// TIA Portal V17 export
// export: Created 2024-09-02T12:50:18.9599664Z, ExportSetting WithDefaults, DisplayName Totally Integrated Automation Portal, DisplayVersion V17, DisplayName TIA Portal Openness, DisplayVersion V17, DisplayName TIA Portal Version Control Interface, DisplayVersion V17, DisplayName STEP 7 Professional, DisplayVersion V17, DisplayName STEP 7 Safety, DisplayVersion V17, DisplayName WinCC Professional, DisplayVersion V17
FUNCTION "AnwFC_Desoutter_OP70_2" : Void   // FC110, LAD
{ S7_Optimized_Access := 'TRUE' }
VERSION : 0.1
// stored: AutoNumber false, IsIECCheckEnabled false, SetENOAutomatically false, UDAEnableTagReadback false
   VAR_TEMP
      tVKE0 : Bool;
      tVKE1 : Bool;
      tAuto : Bool;
      tHand : Bool;
      Motion_Release : Bool;
      t_dummy : Bool;
      tHmiBld : Bool;
      tHmiEnbl : Bool;
      tProgram_nr : Byte;
      tCnt : Int;
      tBAmode : Int;
      tHmiNr : Int;
      tArray_ID_POP : Array[0..15] of Char;
      Part_ID_Ready : Bool;
      tCnt_char : UInt;
      Position_of_ScrewDriver_Ready : Bool;
      tHmiScreen : Bool;
      tHmiRelease : Bool;
   END_VAR
   VAR_TEMP   // added for the SCL form of the ladder/FBD networks
      _w1 : Bool;
      _w2 : Bool;
   END_VAR
BEGIN

REGION Network 1: ############# Start Up Conditions ###############
END_REGION

REGION Network 2: VKE0/1
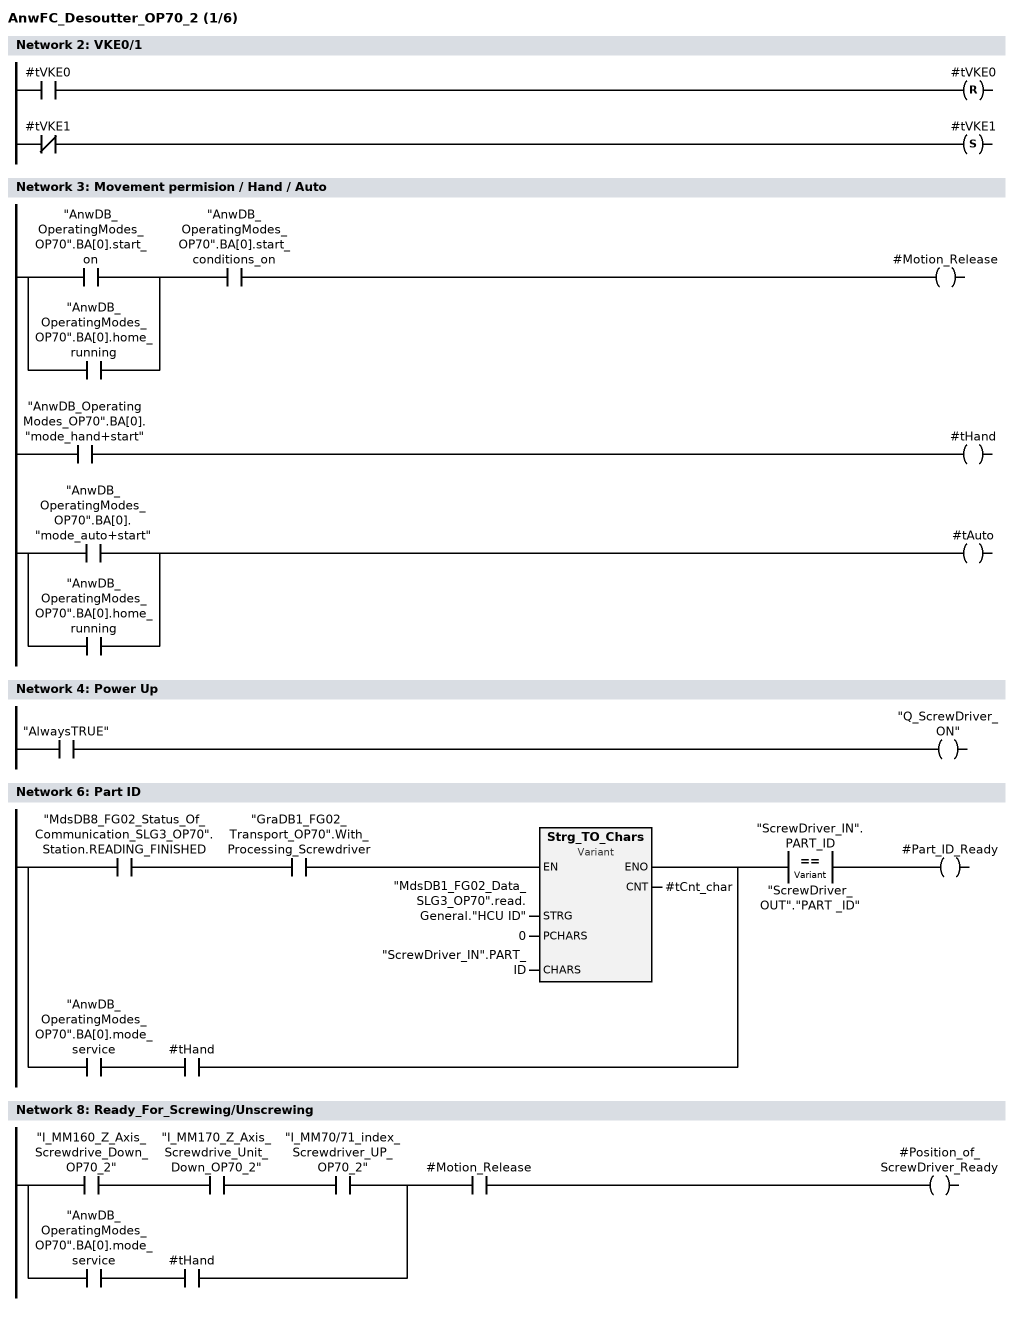
   RUNG wire#powerrail
      Contact( #tVKE0 )
      R_Coil( #tVKE0 )
   END_RUNG
   RUNG wire#powerrail
      I_Contact( #tVKE1 )
      S_Coil( #tVKE1 )
   END_RUNG
   // the same network as SCL:
   IF #tVKE0 THEN #tVKE0 := FALSE; END_IF;
   IF NOT #tVKE1 THEN #tVKE1 := TRUE; END_IF;
END_REGION

REGION Network 3: Movement permision / Hand / Auto
   RUNG wire#powerrail
      Contact( "AnwDB_OperatingModes_OP70".BA[0].start_on )
      wire#w1
      Contact( "AnwDB_OperatingModes_OP70".BA[0].start_conditions_on )
      Coil( #Motion_Release )
   END_RUNG
   RUNG wire#powerrail
      Contact( "AnwDB_OperatingModes_OP70".BA[0].home_running )
   END_RUNG wire#w1
   RUNG wire#powerrail
      Contact( "AnwDB_OperatingModes_OP70".BA[0]."mode_hand+start" )
      Coil( #tHand )
   END_RUNG
   RUNG wire#powerrail
      Contact( "AnwDB_OperatingModes_OP70".BA[0]."mode_auto+start" )
      wire#w2
      Coil( #tAuto )
   END_RUNG
   RUNG wire#powerrail
      Contact( "AnwDB_OperatingModes_OP70".BA[0].home_running )
   END_RUNG wire#w2
   // the same network as SCL:
   #Motion_Release := ("AnwDB_OperatingModes_OP70".BA[0].start_on OR "AnwDB_OperatingModes_OP70".BA[0].home_running) AND "AnwDB_OperatingModes_OP70".BA[0].start_conditions_on;
   #tHand := "AnwDB_OperatingModes_OP70".BA[0]."mode_hand+start";
   #tAuto := "AnwDB_OperatingModes_OP70".BA[0]."mode_auto+start" OR "AnwDB_OperatingModes_OP70".BA[0].home_running;
END_REGION

REGION Network 4: Power Up
   RUNG wire#powerrail
      Contact( "AlwaysTRUE" )
      Coil( "Q_ScrewDriver_ON" )
   END_RUNG
   // the same network as SCL:
   "Q_ScrewDriver_ON" := "AlwaysTRUE";
END_REGION

REGION Network 5: ############# Data Operation ###############
END_REGION

REGION Network 6: Part ID
   RUNG wire#powerrail
      Contact( "MdsDB8_FG02_Status_Of_Communication_SLG3_OP70".Station.READING_FINISHED )
      Contact( "GraDB1_FG02_Transport_OP70".With_Processing_Screwdriver )
      { S7_Templates := "[ptr_type := Variant, strg_type := String]" } Strg_TO_Chars(Strg := "MdsDB1_FG02_Data_SLG3_OP70".read.General."HCU ID", pChars := 0, Chars := "ScrewDriver_IN".PART_ID, Cnt => #tCnt_char)
      wire#w1
      { S7_Templates := "SrcType := Variant" } EQ_Contact(in1 := "ScrewDriver_IN".PART_ID, in2 := "ScrewDriver_OUT"."PART _ID")
      Coil( #Part_ID_Ready )
   END_RUNG
   RUNG wire#powerrail
      Contact( "AnwDB_OperatingModes_OP70".BA[0].mode_service )
      Contact( #tHand )
   END_RUNG wire#w1
   // the same network as SCL:
   #_w1 := "MdsDB8_FG02_Status_Of_Communication_SLG3_OP70".Station.READING_FINISHED AND "GraDB1_FG02_Transport_OP70".With_Processing_Screwdriver;
   Strg_TO_Chars(EN := #_w1,
                 Strg := "MdsDB1_FG02_Data_SLG3_OP70".read.General."HCU ID",
                 pChars := 0,
                 Chars := "ScrewDriver_IN".PART_ID,
                 Cnt => #tCnt_char,
                 ENO => #_w2);
   #Part_ID_Ready := (#_w2 OR ("AnwDB_OperatingModes_OP70".BA[0].mode_service AND #tHand)) AND ("ScrewDriver_IN".PART_ID = "ScrewDriver_OUT"."PART _ID");
END_REGION

REGION Network 7: ############# Program Selection And Start ###############
END_REGION

REGION Network 8: Ready_For_Screwing/Unscrewing
   RUNG wire#powerrail
      Contact( "I_MM160_Z_Axis_Screwdrive_Down_OP70_2" )
      Contact( "I_MM170_Z_Axis_Screwdrive_Unit_Down_OP70_2" )
      Contact( "I_MM70/71_index_Screwdriver_UP_OP70_2" )
      wire#w1
      Contact( #Motion_Release )
      Coil( #Position_of_ScrewDriver_Ready )
   END_RUNG
   RUNG wire#powerrail
      Contact( "AnwDB_OperatingModes_OP70".BA[0].mode_service )
      Contact( #tHand )
   END_RUNG wire#w1
   // the same network as SCL:
   #Position_of_ScrewDriver_Ready := (("I_MM160_Z_Axis_Screwdrive_Down_OP70_2" AND "I_MM170_Z_Axis_Screwdrive_Unit_Down_OP70_2" AND "I_MM70/71_index_Screwdriver_UP_OP70_2") OR ("AnwDB_OperatingModes_OP70".BA[0].mode_service AND #tHand)) AND #Motion_Release;
END_REGION

REGION Network 9: Reset
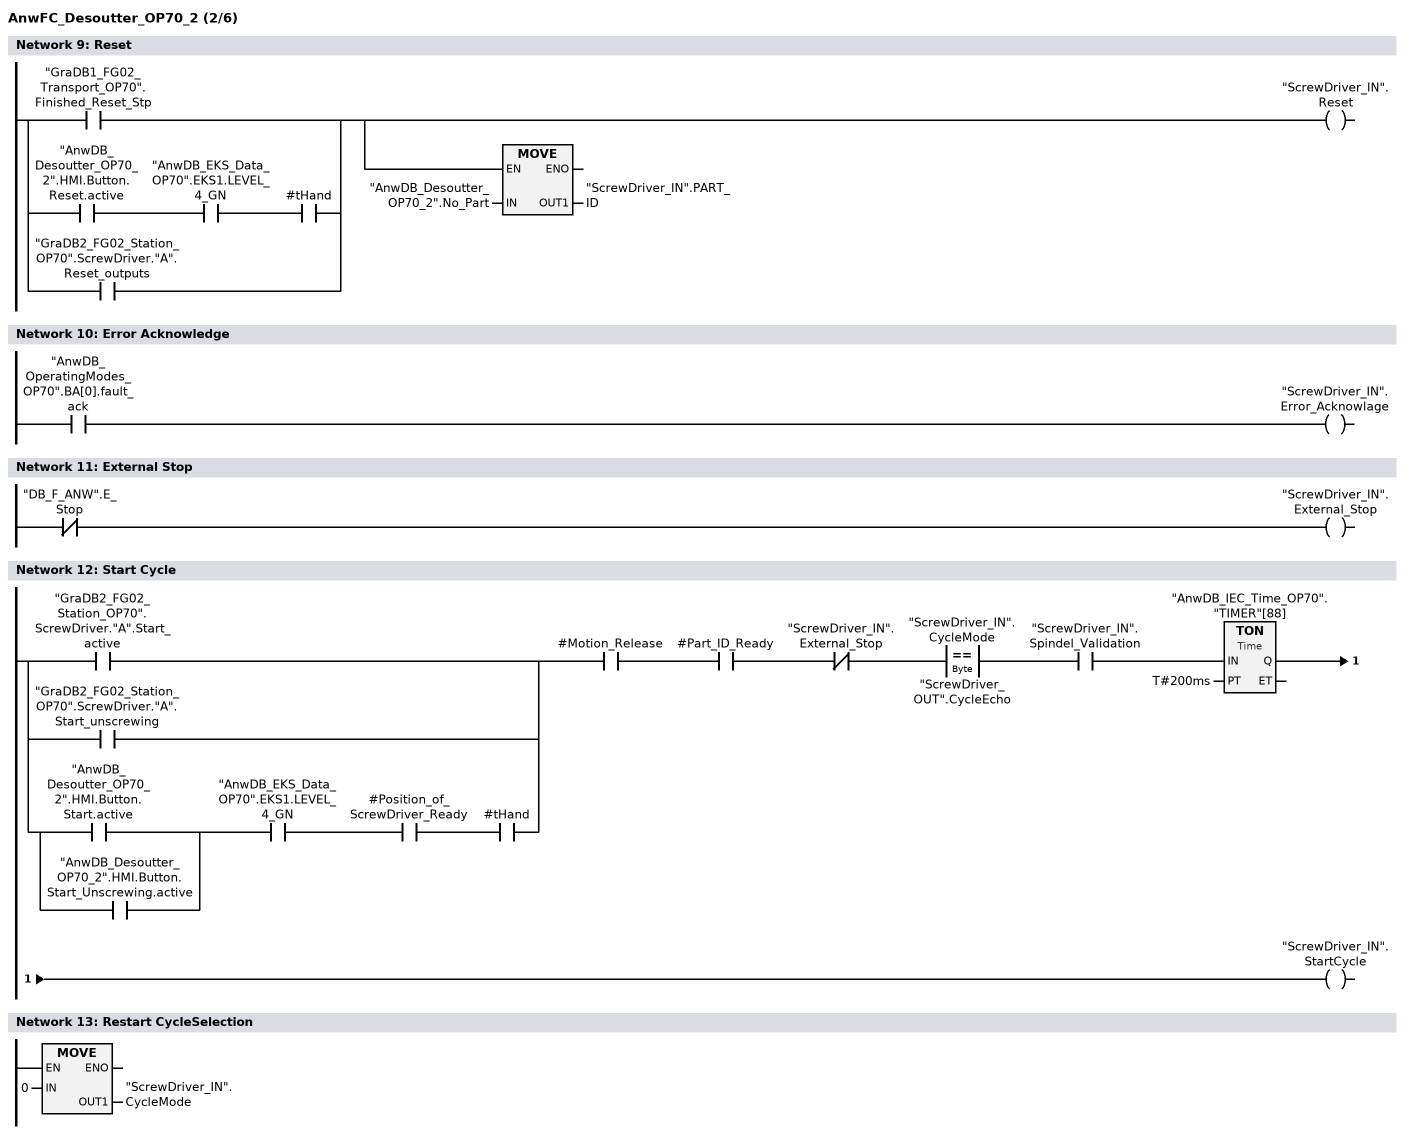
   RUNG wire#powerrail
      Contact( "GraDB1_FG02_Transport_OP70".Finished_Reset_Stp )
      wire#w1
      Coil( "ScrewDriver_IN".Reset )
   END_RUNG
   RUNG wire#powerrail
      Contact( "AnwDB_Desoutter_OP70_2".HMI.Button.Reset.active )
      Contact( "AnwDB_EKS_Data_OP70".EKS1.LEVEL_4_GN )
      Contact( #tHand )
   END_RUNG wire#w1
   RUNG wire#powerrail
      Contact( "GraDB2_FG02_Station_OP70".ScrewDriver."A".Reset_outputs )
   END_RUNG wire#w1
   RUNG wire#w1
      Move(in := "AnwDB_Desoutter_OP70_2".No_Part, out1 => "ScrewDriver_IN".PART_ID)
   END_RUNG
   // the same network as SCL:
   "ScrewDriver_IN".Reset := "GraDB1_FG02_Transport_OP70".Finished_Reset_Stp OR ("AnwDB_Desoutter_OP70_2".HMI.Button.Reset.active AND "AnwDB_EKS_Data_OP70".EKS1.LEVEL_4_GN AND #tHand) OR "GraDB2_FG02_Station_OP70".ScrewDriver."A".Reset_outputs;
   IF "ScrewDriver_IN".Reset THEN "ScrewDriver_IN".PART_ID := "AnwDB_Desoutter_OP70_2".No_Part; END_IF;
END_REGION

REGION Network 10: Error Acknowledge
   RUNG wire#powerrail
      Contact( "AnwDB_OperatingModes_OP70".BA[0].fault_ack )
      Coil( "ScrewDriver_IN".Error_Acknowlage )
   END_RUNG
   // the same network as SCL:
   "ScrewDriver_IN".Error_Acknowlage := "AnwDB_OperatingModes_OP70".BA[0].fault_ack;
END_REGION

REGION Network 11: External Stop
   RUNG wire#powerrail
      I_Contact( "DB_F_ANW".E_Stop )
      Coil( "ScrewDriver_IN".External_Stop )
   END_RUNG
   // the same network as SCL:
   "ScrewDriver_IN".External_Stop := NOT "DB_F_ANW".E_Stop;
END_REGION

REGION Network 12: Start Cycle
   RUNG wire#powerrail
      Contact( "GraDB2_FG02_Station_OP70".ScrewDriver."A".Start_active )
      wire#w1
      Contact( #Motion_Release )
      Contact( #Part_ID_Ready )
      I_Contact( "ScrewDriver_IN".External_Stop )
      { S7_Templates := "SrcType := Byte" } EQ_Contact(in1 := "ScrewDriver_IN".CycleMode, in2 := "ScrewDriver_OUT".CycleEcho)
      Contact( "ScrewDriver_IN".Spindel_Validation )
      { S7_Templates := "time_type := Time" } "AnwDB_IEC_Time_OP70"."TIMER"[88].TON(pt := T#200ms, et =>)
      Coil( "ScrewDriver_IN".StartCycle )
   END_RUNG
   RUNG wire#powerrail
      Contact( "GraDB2_FG02_Station_OP70".ScrewDriver."A".Start_unscrewing )
   END_RUNG wire#w1
   RUNG wire#powerrail
      Contact( "AnwDB_Desoutter_OP70_2".HMI.Button.Start.active )
      wire#w2
      Contact( "AnwDB_EKS_Data_OP70".EKS1.LEVEL_4_GN )
      Contact( #Position_of_ScrewDriver_Ready )
      Contact( #tHand )
   END_RUNG wire#w1
   RUNG wire#powerrail
      Contact( "AnwDB_Desoutter_OP70_2".HMI.Button.Start_Unscrewing.active )
   END_RUNG wire#w2
   // the same network as SCL:
   "AnwDB_IEC_Time_OP70"."TIMER"[88].TON(IN := ("GraDB2_FG02_Station_OP70".ScrewDriver."A".Start_active OR "GraDB2_FG02_Station_OP70".ScrewDriver."A".Start_unscrewing OR (("AnwDB_Desoutter_OP70_2".HMI.Button.Start.active OR "AnwDB_Desoutter_OP70_2".HMI.Button.Start_Unscrewing.active) AND "AnwDB_EKS_Data_OP70".EKS1.LEVEL_4_GN AND #Position_of_ScrewDriver_Ready AND #tHand)) AND #Motion_Release AND #Part_ID_Ready AND NOT "ScrewDriver_IN".External_Stop AND ("ScrewDriver_IN".CycleMode = "ScrewDriver_OUT".CycleEcho) AND "ScrewDriver_IN".Spindel_Validation,
                           PT := T#200ms);
   "ScrewDriver_IN".StartCycle := "AnwDB_IEC_Time_OP70"."TIMER"[88].Q;
END_REGION

REGION Network 13: Restart CycleSelection
   RUNG wire#powerrail
      Move(in := 0, out1 => "ScrewDriver_IN".CycleMode)
   END_RUNG
   // the same network as SCL:
   "ScrewDriver_IN".CycleMode := 0;
END_REGION

REGION Network 14: Cycle Selection - Hand
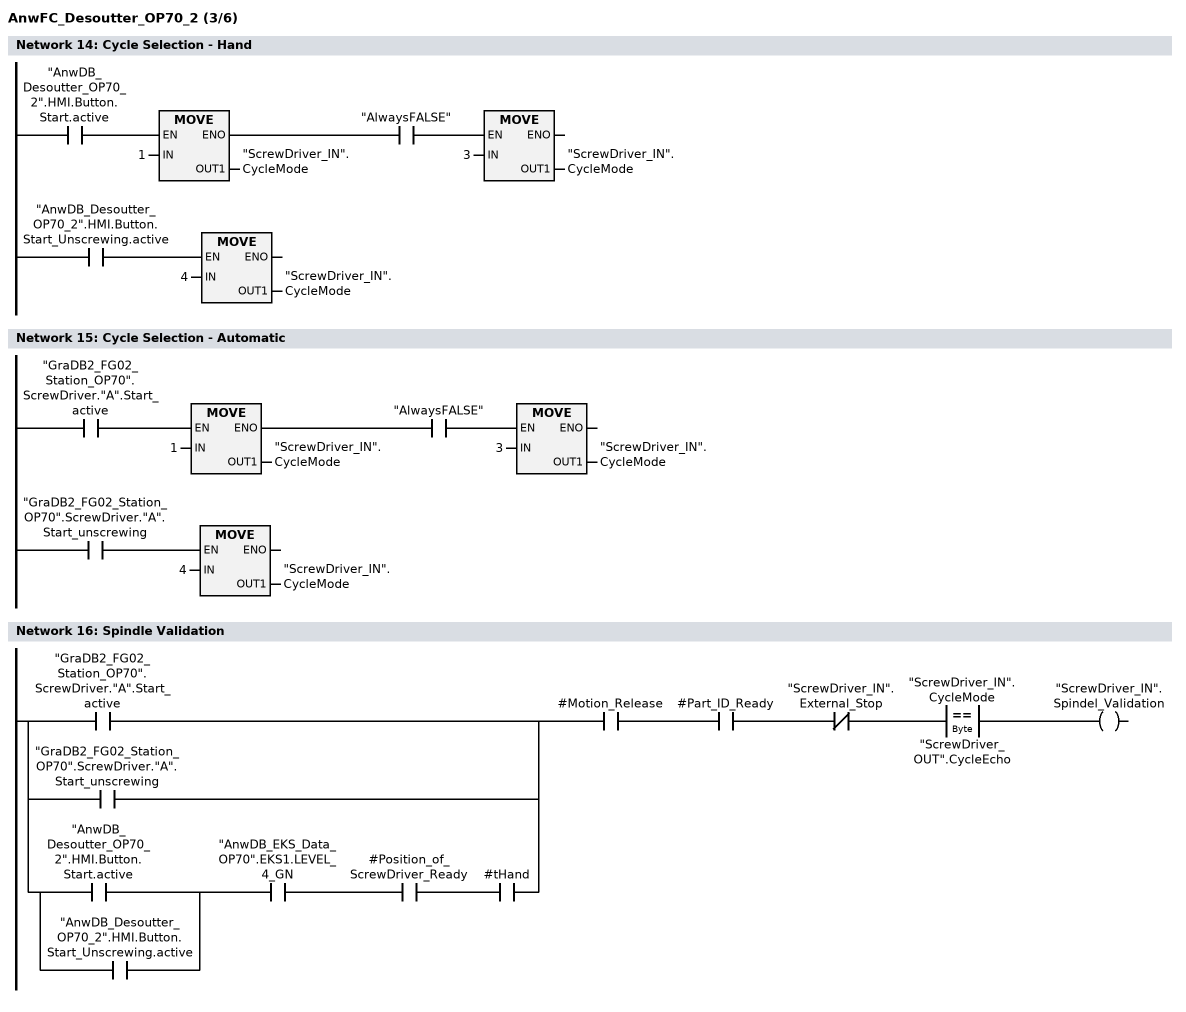
   RUNG wire#powerrail
      Contact( "AnwDB_Desoutter_OP70_2".HMI.Button.Start.active )
      Move(in := 1, out1 => "ScrewDriver_IN".CycleMode)
      Contact( "AlwaysFALSE" )
      Move(in := 3, out1 => "ScrewDriver_IN".CycleMode)
   END_RUNG
   RUNG wire#powerrail
      Contact( "AnwDB_Desoutter_OP70_2".HMI.Button.Start_Unscrewing.active )
      Move(in := 4, out1 => "ScrewDriver_IN".CycleMode)
   END_RUNG
   // the same network as SCL:
   IF "AnwDB_Desoutter_OP70_2".HMI.Button.Start.active THEN "ScrewDriver_IN".CycleMode := 1; END_IF;
   IF "AnwDB_Desoutter_OP70_2".HMI.Button.Start.active AND "AlwaysFALSE" THEN
       "ScrewDriver_IN".CycleMode := 3;
   END_IF;
   IF "AnwDB_Desoutter_OP70_2".HMI.Button.Start_Unscrewing.active THEN
       "ScrewDriver_IN".CycleMode := 4;
   END_IF;
END_REGION

REGION Network 15: Cycle Selection - Automatic
   RUNG wire#powerrail
      Contact( "GraDB2_FG02_Station_OP70".ScrewDriver."A".Start_active )
      Move(in := 1, out1 => "ScrewDriver_IN".CycleMode)
      Contact( "AlwaysFALSE" )
      Move(in := 3, out1 => "ScrewDriver_IN".CycleMode)
   END_RUNG
   RUNG wire#powerrail
      Contact( "GraDB2_FG02_Station_OP70".ScrewDriver."A".Start_unscrewing )
      Move(in := 4, out1 => "ScrewDriver_IN".CycleMode)
   END_RUNG
   // the same network as SCL:
   IF "GraDB2_FG02_Station_OP70".ScrewDriver."A".Start_active THEN "ScrewDriver_IN".CycleMode := 1; END_IF;
   IF "GraDB2_FG02_Station_OP70".ScrewDriver."A".Start_active AND "AlwaysFALSE" THEN
       "ScrewDriver_IN".CycleMode := 3;
   END_IF;
   IF "GraDB2_FG02_Station_OP70".ScrewDriver."A".Start_unscrewing THEN
       "ScrewDriver_IN".CycleMode := 4;
   END_IF;
END_REGION

REGION Network 16: Spindle Validation
   RUNG wire#powerrail
      Contact( "GraDB2_FG02_Station_OP70".ScrewDriver."A".Start_active )
      wire#w1
      Contact( #Motion_Release )
      Contact( #Part_ID_Ready )
      I_Contact( "ScrewDriver_IN".External_Stop )
      { S7_Templates := "SrcType := Byte" } EQ_Contact(in1 := "ScrewDriver_IN".CycleMode, in2 := "ScrewDriver_OUT".CycleEcho)
      Coil( "ScrewDriver_IN".Spindel_Validation )
   END_RUNG
   RUNG wire#powerrail
      Contact( "GraDB2_FG02_Station_OP70".ScrewDriver."A".Start_unscrewing )
   END_RUNG wire#w1
   RUNG wire#powerrail
      Contact( "AnwDB_Desoutter_OP70_2".HMI.Button.Start.active )
      wire#w2
      Contact( "AnwDB_EKS_Data_OP70".EKS1.LEVEL_4_GN )
      Contact( #Position_of_ScrewDriver_Ready )
      Contact( #tHand )
   END_RUNG wire#w1
   RUNG wire#powerrail
      Contact( "AnwDB_Desoutter_OP70_2".HMI.Button.Start_Unscrewing.active )
   END_RUNG wire#w2
   // the same network as SCL:
   "ScrewDriver_IN".Spindel_Validation := ("GraDB2_FG02_Station_OP70".ScrewDriver."A".Start_active OR "GraDB2_FG02_Station_OP70".ScrewDriver."A".Start_unscrewing OR (("AnwDB_Desoutter_OP70_2".HMI.Button.Start.active OR "AnwDB_Desoutter_OP70_2".HMI.Button.Start_Unscrewing.active) AND "AnwDB_EKS_Data_OP70".EKS1.LEVEL_4_GN AND #Position_of_ScrewDriver_Ready AND #tHand)) AND #Motion_Release AND #Part_ID_Ready AND NOT "ScrewDriver_IN".External_Stop AND ("ScrewDriver_IN".CycleMode = "ScrewDriver_OUT".CycleEcho);
END_REGION

REGION Network 17: ############# Program Status ###############
END_REGION

REGION Network 18: BEA[3].Ebit[1] - / BEA[3].Ebit[1] - Searching Program
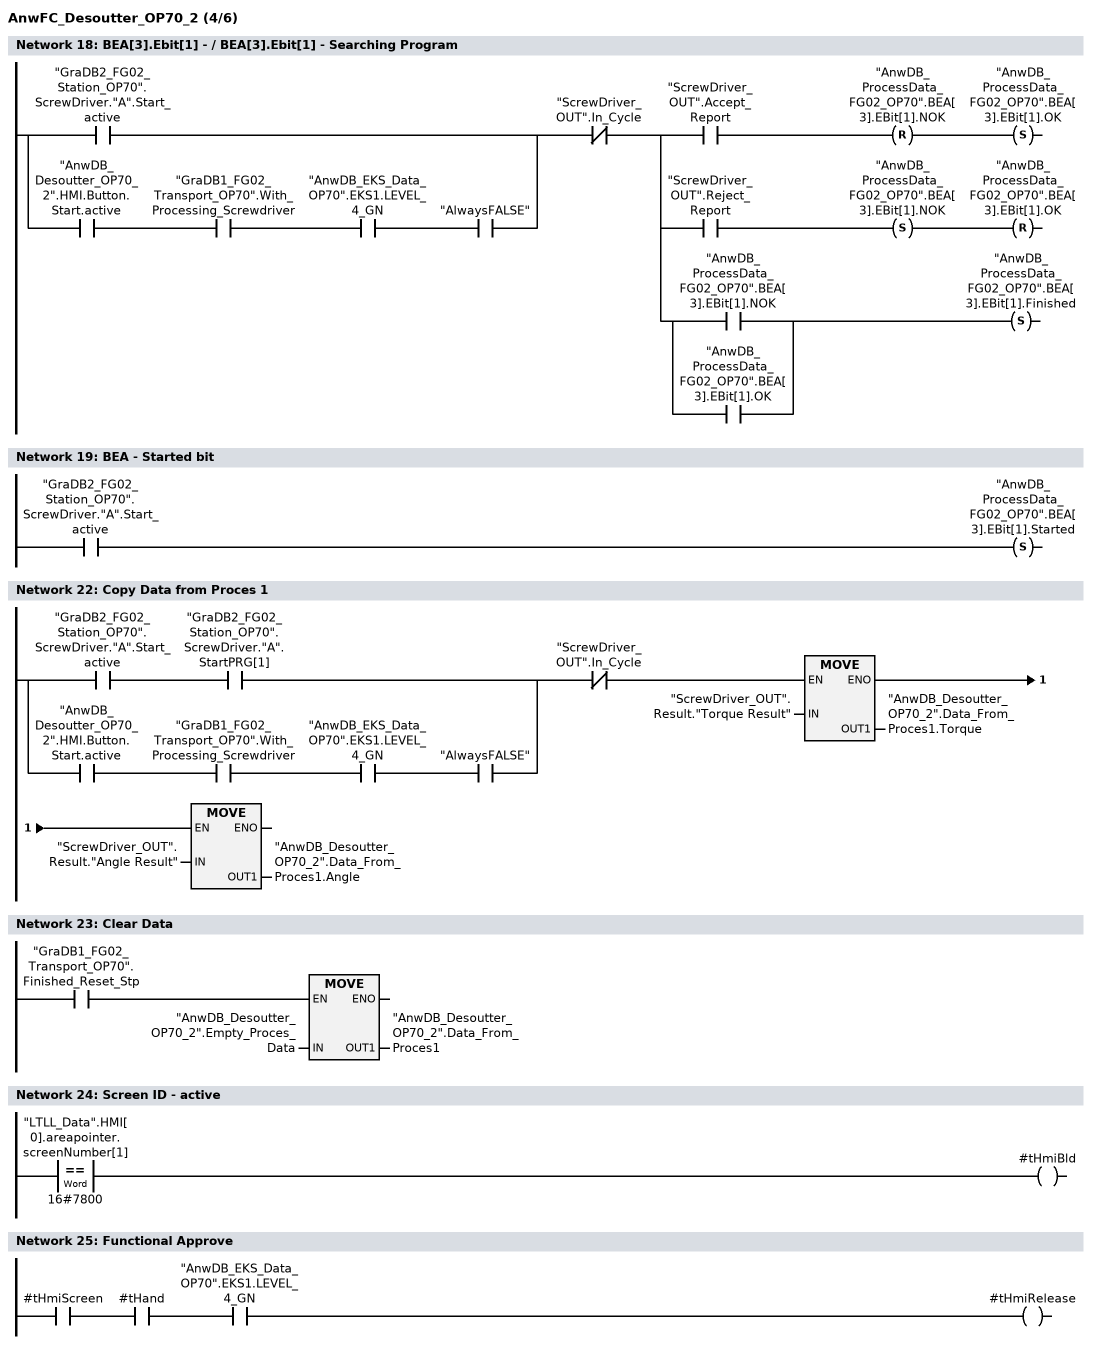
   RUNG wire#powerrail
      Contact( "GraDB2_FG02_Station_OP70".ScrewDriver."A".Start_active )
      wire#w1
      I_Contact( "ScrewDriver_OUT".In_Cycle )
      wire#w2
      Contact( "ScrewDriver_OUT".Accept_Report )
      R_Coil( "AnwDB_ProcessData_FG02_OP70".BEA[3].EBit[1].NOK )
      S_Coil( "AnwDB_ProcessData_FG02_OP70".BEA[3].EBit[1].OK )
   END_RUNG
   RUNG wire#powerrail
      Contact( "AnwDB_Desoutter_OP70_2".HMI.Button.Start.active )
      Contact( "GraDB1_FG02_Transport_OP70".With_Processing_Screwdriver )
      Contact( "AnwDB_EKS_Data_OP70".EKS1.LEVEL_4_GN )
      Contact( "AlwaysFALSE" )
   END_RUNG wire#w1
   RUNG wire#w2
      Contact( "ScrewDriver_OUT".Reject_Report )
      S_Coil( "AnwDB_ProcessData_FG02_OP70".BEA[3].EBit[1].NOK )
      R_Coil( "AnwDB_ProcessData_FG02_OP70".BEA[3].EBit[1].OK )
   END_RUNG
   RUNG wire#w2
      Contact( "AnwDB_ProcessData_FG02_OP70".BEA[3].EBit[1].NOK )
      wire#w3
      S_Coil( "AnwDB_ProcessData_FG02_OP70".BEA[3].EBit[1].Finished )
   END_RUNG
   RUNG wire#w2
      Contact( "AnwDB_ProcessData_FG02_OP70".BEA[3].EBit[1].OK )
   END_RUNG wire#w3
   // the same network as SCL:
   #_w1 := ("GraDB2_FG02_Station_OP70".ScrewDriver."A".Start_active OR ("AnwDB_Desoutter_OP70_2".HMI.Button.Start.active AND "GraDB1_FG02_Transport_OP70".With_Processing_Screwdriver AND "AnwDB_EKS_Data_OP70".EKS1.LEVEL_4_GN AND "AlwaysFALSE")) AND NOT "ScrewDriver_OUT".In_Cycle;
   IF #_w1 AND "ScrewDriver_OUT".Accept_Report THEN
       "AnwDB_ProcessData_FG02_OP70".BEA[3].EBit[1].NOK := FALSE;
       "AnwDB_ProcessData_FG02_OP70".BEA[3].EBit[1].OK := TRUE;
   END_IF;
   IF #_w1 AND "ScrewDriver_OUT".Reject_Report THEN
       "AnwDB_ProcessData_FG02_OP70".BEA[3].EBit[1].NOK := TRUE;
       "AnwDB_ProcessData_FG02_OP70".BEA[3].EBit[1].OK := FALSE;
   END_IF;
   IF #_w1 AND ("AnwDB_ProcessData_FG02_OP70".BEA[3].EBit[1].NOK OR "AnwDB_ProcessData_FG02_OP70".BEA[3].EBit[1].OK) THEN
       "AnwDB_ProcessData_FG02_OP70".BEA[3].EBit[1].Finished := TRUE;
   END_IF;
END_REGION

REGION Network 19: BEA - Started bit
   RUNG wire#powerrail
      Contact( "GraDB2_FG02_Station_OP70".ScrewDriver."A".Start_active )
      S_Coil( "AnwDB_ProcessData_FG02_OP70".BEA[3].EBit[1].Started )
   END_RUNG
   // the same network as SCL:
   IF "GraDB2_FG02_Station_OP70".ScrewDriver."A".Start_active THEN
       "AnwDB_ProcessData_FG02_OP70".BEA[3].EBit[1].Started := TRUE;
   END_IF;
END_REGION

REGION Network 20: ############# HMI ###############
END_REGION

REGION Network 21: ############# Data Copy ###############
END_REGION

REGION Network 22: Copy Data from Proces 1
   RUNG wire#powerrail
      Contact( "GraDB2_FG02_Station_OP70".ScrewDriver."A".Start_active )
      Contact( "GraDB2_FG02_Station_OP70".ScrewDriver."A".StartPRG[1] )
      wire#w1
      I_Contact( "ScrewDriver_OUT".In_Cycle )
      Move(in := "ScrewDriver_OUT".Result."Torque Result", out1 => "AnwDB_Desoutter_OP70_2".Data_From_Proces1.Torque)
      Move(in := "ScrewDriver_OUT".Result."Angle Result", out1 => "AnwDB_Desoutter_OP70_2".Data_From_Proces1.Angle)
   END_RUNG
   RUNG wire#powerrail
      Contact( "AnwDB_Desoutter_OP70_2".HMI.Button.Start.active )
      Contact( "GraDB1_FG02_Transport_OP70".With_Processing_Screwdriver )
      Contact( "AnwDB_EKS_Data_OP70".EKS1.LEVEL_4_GN )
      Contact( "AlwaysFALSE" )
   END_RUNG wire#w1
   // the same network as SCL:
   IF (("GraDB2_FG02_Station_OP70".ScrewDriver."A".Start_active AND "GraDB2_FG02_Station_OP70".ScrewDriver."A".StartPRG[1]) OR ("AnwDB_Desoutter_OP70_2".HMI.Button.Start.active AND "GraDB1_FG02_Transport_OP70".With_Processing_Screwdriver AND "AnwDB_EKS_Data_OP70".EKS1.LEVEL_4_GN AND "AlwaysFALSE")) AND NOT "ScrewDriver_OUT".In_Cycle THEN
       "AnwDB_Desoutter_OP70_2".Data_From_Proces1.Torque := "ScrewDriver_OUT".Result."Torque Result";
       "AnwDB_Desoutter_OP70_2".Data_From_Proces1.Angle := "ScrewDriver_OUT".Result."Angle Result";
   END_IF;
END_REGION

REGION Network 23: Clear Data
   RUNG wire#powerrail
      Contact( "GraDB1_FG02_Transport_OP70".Finished_Reset_Stp )
      Move(in := "AnwDB_Desoutter_OP70_2".Empty_Proces_Data, out1 => "AnwDB_Desoutter_OP70_2".Data_From_Proces1)
   END_RUNG
   // the same network as SCL:
   IF "GraDB1_FG02_Transport_OP70".Finished_Reset_Stp THEN
       "AnwDB_Desoutter_OP70_2".Data_From_Proces1 := "AnwDB_Desoutter_OP70_2".Empty_Proces_Data;
   END_IF;
END_REGION

REGION Network 24: Screen ID - active
   RUNG wire#powerrail
      { S7_Templates := "SrcType := Word" } EQ_Contact(in1 := "LTLL_Data".HMI[0].areapointer.screenNumber[1], in2 := 16#7800)
      Coil( #tHmiBld )
   END_RUNG
   // the same network as SCL:
   #tHmiBld := "LTLL_Data".HMI[0].areapointer.screenNumber[1] = 16#7800;
END_REGION

REGION Network 25: Functional Approve
   RUNG wire#powerrail
      Contact( #tHmiScreen )
      Contact( #tHand )
      Contact( "AnwDB_EKS_Data_OP70".EKS1.LEVEL_4_GN )
      Coil( #tHmiRelease )
   END_RUNG
   // the same network as SCL:
   #tHmiRelease := #tHmiScreen AND #tHand AND "AnwDB_EKS_Data_OP70".EKS1.LEVEL_4_GN;
END_REGION

REGION Network 26: Available of Button
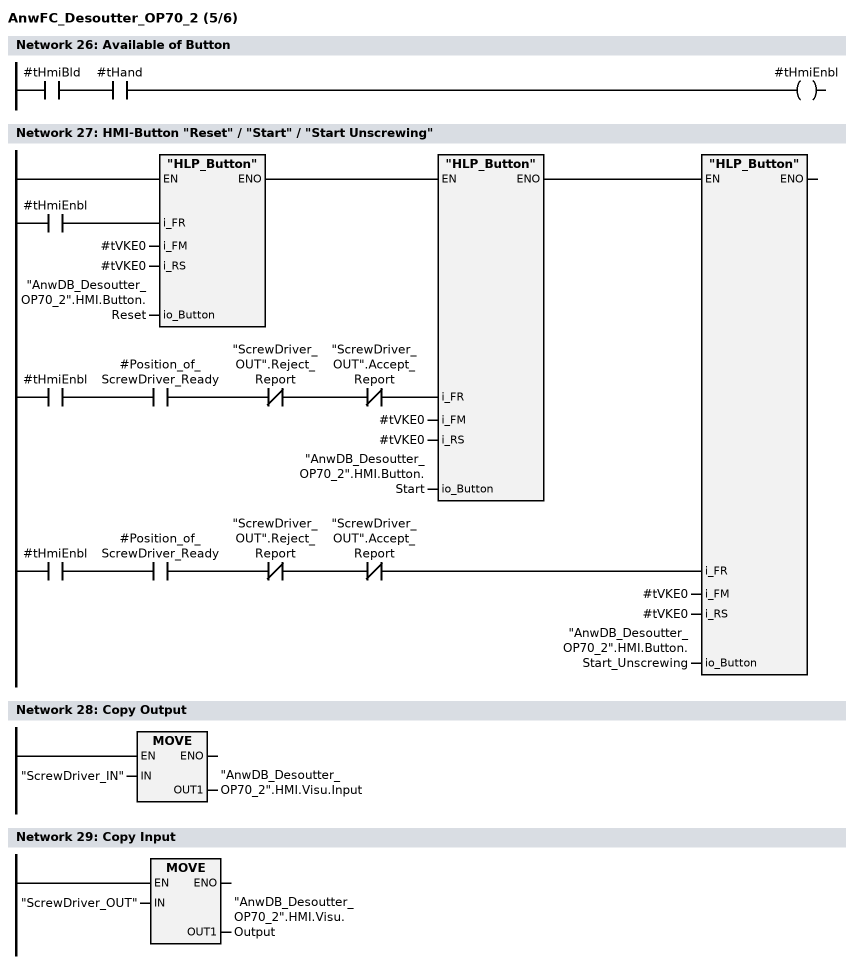
   RUNG wire#powerrail
      Contact( #tHmiBld )
      Contact( #tHand )
      Coil( #tHmiEnbl )
   END_RUNG
   // the same network as SCL:
   #tHmiEnbl := #tHmiBld AND #tHand;
END_REGION

REGION Network 27: HMI-Button "Reset" / "Start" / "Start Unscrewing"
   RUNG wire#powerrail
      "HLP_Button"(i_FR := wire#w1, i_FM := #tVKE0, i_RS := #tVKE0, io_Button := "AnwDB_Desoutter_OP70_2".HMI.Button.Reset)
      "HLP_Button"(i_FR := wire#w2, i_FM := #tVKE0, i_RS := #tVKE0, io_Button := "AnwDB_Desoutter_OP70_2".HMI.Button.Start)
      "HLP_Button"(i_FR := wire#w3, i_FM := #tVKE0, i_RS := #tVKE0, io_Button := "AnwDB_Desoutter_OP70_2".HMI.Button.Start_Unscrewing)
   END_RUNG
   RUNG wire#powerrail
      Contact( #tHmiEnbl )
   END_RUNG wire#w1
   RUNG wire#powerrail
      Contact( #tHmiEnbl )
      Contact( #Position_of_ScrewDriver_Ready )
      I_Contact( "ScrewDriver_OUT".Reject_Report )
      I_Contact( "ScrewDriver_OUT".Accept_Report )
   END_RUNG wire#w2
   RUNG wire#powerrail
      Contact( #tHmiEnbl )
      Contact( #Position_of_ScrewDriver_Ready )
      I_Contact( "ScrewDriver_OUT".Reject_Report )
      I_Contact( "ScrewDriver_OUT".Accept_Report )
   END_RUNG wire#w3
   // the same network as SCL:
   "HLP_Button"(i_FR := #tHmiEnbl,
                i_FM := #tVKE0,
                i_RS := #tVKE0,
                io_Button := "AnwDB_Desoutter_OP70_2".HMI.Button.Reset,
                ENO => #_w1);
   "HLP_Button"(EN := #_w1,
                i_FR := #tHmiEnbl AND #Position_of_ScrewDriver_Ready AND NOT "ScrewDriver_OUT".Reject_Report AND NOT "ScrewDriver_OUT".Accept_Report,
                i_FM := #tVKE0,
                i_RS := #tVKE0,
                io_Button := "AnwDB_Desoutter_OP70_2".HMI.Button.Start,
                ENO => #_w2);
   IF #_w2 THEN
       "HLP_Button"(i_FR := #tHmiEnbl AND #Position_of_ScrewDriver_Ready AND NOT "ScrewDriver_OUT".Reject_Report AND NOT "ScrewDriver_OUT".Accept_Report,
                    i_FM := #tVKE0,
                    i_RS := #tVKE0,
                    io_Button := "AnwDB_Desoutter_OP70_2".HMI.Button.Start_Unscrewing);
   END_IF;
END_REGION

REGION Network 28: Copy Output
   RUNG wire#powerrail
      Move(in := "ScrewDriver_IN", out1 => "AnwDB_Desoutter_OP70_2".HMI.Visu.Input)
   END_RUNG
   // the same network as SCL:
   "AnwDB_Desoutter_OP70_2".HMI.Visu.Input := "ScrewDriver_IN";
END_REGION

REGION Network 29: Copy Input
   RUNG wire#powerrail
      Move(in := "ScrewDriver_OUT", out1 => "AnwDB_Desoutter_OP70_2".HMI.Visu.Output)
   END_RUNG
   // the same network as SCL:
   "AnwDB_Desoutter_OP70_2".HMI.Visu.Output := "ScrewDriver_OUT";
END_REGION

REGION Network 30: Select program / Copy Output
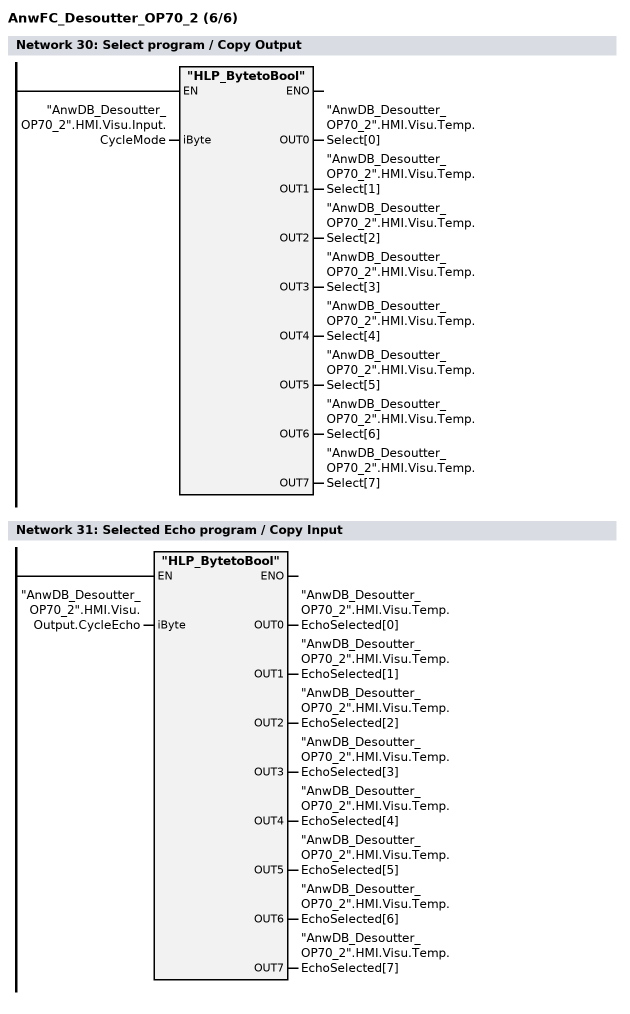
   RUNG wire#powerrail
      "HLP_BytetoBool"(iByte := "AnwDB_Desoutter_OP70_2".HMI.Visu.Input.CycleMode, OUT0 => "AnwDB_Desoutter_OP70_2".HMI.Visu.Temp.Select[0], OUT1 => "AnwDB_Desoutter_OP70_2".HMI.Visu.Temp.Select[1], OUT2 => "AnwDB_Desoutter_OP70_2".HMI.Visu.Temp.Select[2], OUT3 => "AnwDB_Desoutter_OP70_2".HMI.Visu.Temp.Select[3], OUT4 => "AnwDB_Desoutter_OP70_2".HMI.Visu.Temp.Select[4], OUT5 => "AnwDB_Desoutter_OP70_2".HMI.Visu.Temp.Select[5], OUT6 => "AnwDB_Desoutter_OP70_2".HMI.Visu.Temp.Select[6], OUT7 => "AnwDB_Desoutter_OP70_2".HMI.Visu.Temp.Select[7])
   END_RUNG
   // the same network as SCL:
   "HLP_BytetoBool"(iByte := "AnwDB_Desoutter_OP70_2".HMI.Visu.Input.CycleMode,
                    OUT0 => "AnwDB_Desoutter_OP70_2".HMI.Visu.Temp.Select[0],
                    OUT1 => "AnwDB_Desoutter_OP70_2".HMI.Visu.Temp.Select[1],
                    OUT2 => "AnwDB_Desoutter_OP70_2".HMI.Visu.Temp.Select[2],
                    OUT3 => "AnwDB_Desoutter_OP70_2".HMI.Visu.Temp.Select[3],
                    OUT4 => "AnwDB_Desoutter_OP70_2".HMI.Visu.Temp.Select[4],
                    OUT5 => "AnwDB_Desoutter_OP70_2".HMI.Visu.Temp.Select[5],
                    OUT6 => "AnwDB_Desoutter_OP70_2".HMI.Visu.Temp.Select[6],
                    OUT7 => "AnwDB_Desoutter_OP70_2".HMI.Visu.Temp.Select[7]);
END_REGION

REGION Network 31: Selected Echo program / Copy Input
   RUNG wire#powerrail
      "HLP_BytetoBool"(iByte := "AnwDB_Desoutter_OP70_2".HMI.Visu.Output.CycleEcho, OUT0 => "AnwDB_Desoutter_OP70_2".HMI.Visu.Temp.EchoSelected[0], OUT1 => "AnwDB_Desoutter_OP70_2".HMI.Visu.Temp.EchoSelected[1], OUT2 => "AnwDB_Desoutter_OP70_2".HMI.Visu.Temp.EchoSelected[2], OUT3 => "AnwDB_Desoutter_OP70_2".HMI.Visu.Temp.EchoSelected[3], OUT4 => "AnwDB_Desoutter_OP70_2".HMI.Visu.Temp.EchoSelected[4], OUT5 => "AnwDB_Desoutter_OP70_2".HMI.Visu.Temp.EchoSelected[5], OUT6 => "AnwDB_Desoutter_OP70_2".HMI.Visu.Temp.EchoSelected[6], OUT7 => "AnwDB_Desoutter_OP70_2".HMI.Visu.Temp.EchoSelected[7])
   END_RUNG
   // the same network as SCL:
   "HLP_BytetoBool"(iByte := "AnwDB_Desoutter_OP70_2".HMI.Visu.Output.CycleEcho,
                    OUT0 => "AnwDB_Desoutter_OP70_2".HMI.Visu.Temp.EchoSelected[0],
                    OUT1 => "AnwDB_Desoutter_OP70_2".HMI.Visu.Temp.EchoSelected[1],
                    OUT2 => "AnwDB_Desoutter_OP70_2".HMI.Visu.Temp.EchoSelected[2],
                    OUT3 => "AnwDB_Desoutter_OP70_2".HMI.Visu.Temp.EchoSelected[3],
                    OUT4 => "AnwDB_Desoutter_OP70_2".HMI.Visu.Temp.EchoSelected[4],
                    OUT5 => "AnwDB_Desoutter_OP70_2".HMI.Visu.Temp.EchoSelected[5],
                    OUT6 => "AnwDB_Desoutter_OP70_2".HMI.Visu.Temp.EchoSelected[6],
                    OUT7 => "AnwDB_Desoutter_OP70_2".HMI.Visu.Temp.EchoSelected[7]);
END_REGION

REGION Network 32 (SCL): Copy Nr of variant to HMI

   IF #Part_ID_Ready THEN
           "AnwDB_Desoutter_OP70_2".HMI.Variant_Number := "MdsDB1_FG02_Data_SLG3_OP70".read.General."HCU ID";
           ;
       ELSE
           "AnwDB_Desoutter_OP70_2".HMI.Variant_Number := 'Error';
       END_IF;
END_REGION
END_FUNCTION
